              if(rq_write_lbp[index] == -1 and rq_read_lbp[index] != -1):
                  rq_write_lbp[index] = rq_read_lbp[index]
                  rq_write_lbp_previous[index] = rq_read_lbp[index]
              elif(rq_write_lbp_previous[index] == -1 and rq_read_lbp[index] != -1):
                  rq_write_lbp_previous[index] = rq_read_lbp[index]
              end

              if(rq_write_lrd[index] == -1 and rq_read_lrd[index] != -1):
                  rq_write_lrd[index] = rq_read_lrd[index]
                  rq_write_lrd_previous[index] = rq_read_lrd[index]
              elif(rq_write_lrd_previous[index] == -1 and rq_read_lrd[index] != -1):
                  rq_write_lrd_previous[index] = rq_read_lrd[index]
              end

              if(rq_write_lbl[index] == -1 and rq_read_lbl[index] != -1):
                  rq_write_lbl[index] = rq_read_lbl[index]
                  rq_write_lbl_previous[index] = rq_read_lbl[index]
              elif(rq_write_lbl_previous[index] == -1 and rq_read_lbl[index] != -1):
                  rq_write_lbl_previous[index] = rq_read_lbl[index]
              end

              if(rq_write_lgn[index] == -1 and rq_read_lgn[index] != -1):
                  rq_write_lgn[index] = rq_read_lgn[index]
                  rq_write_lgn_previous[index] = rq_read_lgn[index]
              elif(rq_write_lgn_previous[index] == -1 and rq_read_lgn[index] != -1):
                  rq_write_lgn_previous[index] = rq_read_lgn[index]
              end

              if(rq_write_msc[index] == -1 and rq_read_msc[index] != -1):
                  rq_write_msc[index] = rq_read_msc[index]
                  rq_write_msc_previous[index] = rq_read_msc[index]
              elif(rq_write_msc_previous[index] == -1 and rq_read_msc[index] != -1):
                  rq_write_msc_previous[index] = rq_read_msc[index]
              end

              if(rq_write_mod[index] == -1 and rq_read_mod[index] != -1):
                  rq_write_mod[index] = rq_read_mod[index]
                  rq_write_mod_previous[index] = rq_read_mod[index]
              elif(rq_write_mod_previous[index] == -1 and rq_read_mod[index] != -1):
                  rq_write_mod_previous[index] = rq_read_mod[index]
              end

          end
          index = index + 1
      end
  end

  def rq_comm_set_var(var, value=0, gripper_socket="1"):
      socket_set_var(var, value, gripper_socket)
      return socket_read_byte_list(3, gripper_socket)
  end

  def rq_comm_set_pos_spe_for(pos=0, speed=0, force=0, gripper_socket="1"):
      socket_send_string("SET POS", gripper_socket)
      socket_send_byte(32, gripper_socket)
      socket_send_string(pos, gripper_socket)
      socket_send_byte(32, gripper_socket)
      socket_send_string("SPE", gripper_socket)
      socket_send_byte(32, gripper_socket)
      socket_send_string(speed, gripper_socket)
      socket_send_byte(32, gripper_socket)
      socket_send_string("FOR", gripper_socket)
      socket_send_byte(32, gripper_socket)
      socket_send_string(force, gripper_socket)
      socket_send_byte(10, gripper_socket)
      return socket_read_byte_list(3, gripper_socket)
  end

  def rq_comm_read_variables():
      index = 0

      while(index <= 3):
          socket = rq_index_to_socket(index)

          if(gripper_connected[index]):

              if(rq_read_act_req[index]):
                  rq_read_act[index] = socket_get_var("ACT", socket)
                  rq_read_act_req[index] = False
              end

              if(rq_read_gto_req[index]):
                  rq_read_gto[index] = socket_get_var("GTO", socket)
                  rq_read_gto_req[index] = False
              end

              if(rq_read_pre_req[index]):
                  rq_read_pre[index] = socket_get_var("PRE", socket)
                  rq_read_pre_req[index] = False
              end

              if(rq_read_pos_req[index]):
                  rq_read_pos[index] = socket_get_var("POS", socket)
                  rq_read_pos_req[index] = False
              end

              if(rq_read_spe_req[index]):
                  rq_read_spe[index] = socket_get_var("SPE", socket)
                  rq_read_spe_req[index] = False
              end

              if(rq_read_for_req[index]):
                  rq_read_for[index] = socket_get_var("FOR", socket)
                  rq_read_for_req[index] = False
              end

              if(rq_read_obj_req[index]):
                  rq_read_obj[index] = socket_get_var("OBJ", socket)
                  rq_read_obj_req[index] = False
              end

              if(rq_read_sta_req[index]):
                  rq_read_sta[index] = socket_get_var("STA", socket)
                  rq_read_sta_req[index] = False
              end

              if(rq_read_mod_req[index]):
                  rq_read_mod[index] = socket_get_var("MOD", socket)
                  rq_read_mod_req[index] = False
              end

              if(rq_read_flt_req[index]):
                  rq_read_flt[index] = socket_get_var("FLT",socket)
                  rq_read_flt_req[index] = False
              end

              if(rq_read_lbp_req[index]):
                  rq_read_lbp[index] = socket_get_var("LBP", socket)
                  rq_read_lbp_req[index] = False
              end

              if(rq_read_lrd_req[index]):
                  rq_read_lrd[index] = socket_get_var("LRD", socket)
                  rq_read_lrd_req[index] = False
              end

              if(rq_read_lbl_req[index]):
                  rq_read_lbl[index] = socket_get_var("LBL",socket)
                  rq_read_lbl_req[index] = False
              end

              if(rq_read_lgn_req[index]):
                  rq_read_lgn[index] = socket_get_var("LGN", socket)
                  rq_read_lgn_req[index] = False
              end

              if(rq_read_msc_req[index]):
                  rq_read_msc[index] = socket_get_var("MSC", socket)
                  rq_read_msc_req[index] = False
              end

              if(rq_read_cou_req[index]):
                  rq_read_cou[index] = socket_get_var("COU", socket)
                  rq_read_cou_req[index] = False
              end

              if(rq_read_ncy_req[index]):
                  rq_read_ncy[index] = socket_get_var("NCY", socket)
                  rq_read_ncy_req[index] = False
              end

              if(rq_read_dst_req[index]):
                  rq_read_dst[index] = socket_get_var("DST", socket)
                  rq_read_dst_req[index] = False
              end

              if(rq_read_pco_req[index]):
                  rq_read_pco[index] = socket_get_var("PCO", socket)
                  rq_read_pco_req[index] = False
              end
          end
          index = index + 1
      end
  end

  def rq_comm_read_constants():

      if(gripper_connected[0]):
          while(rq_read_snu_1 == rq_string_initial_value):
              socket_send_string("GET SNU", "1")
              rq_read_snu_1 = socket_read_string("1")
          end

          while(rq_read_fwv_1 == rq_string_initial_value):
              socket_send_string("GET FWV", "1")
              rq_read_fwv_1 = socket_read_string("1")
          end

          while(rq_read_ver_1 == rq_string_initial_value):
              socket_send_string("GET VER", "1")
              rq_read_ver_1 = socket_read_string("1")
          end
      end

      if(gripper_connected[1]):
          while(rq_read_snu_2 == rq_string_initial_value):
              socket_send_string("GET SNU", "2")
              rq_read_snu_2 = socket_read_string("2")
          end

          while(rq_read_fwv_2 == rq_string_initial_value):
              socket_send_string("GET FWV", "2")
              rq_read_fwv_2 = socket_read_string("2")
          end

          while(rq_read_ver_2 == rq_string_initial_value):
              socket_send_string("GET VER", "2")
              rq_read_ver_2 = socket_read_string("2")
          end
      end

      if(gripper_connected[2]):
          while(rq_read_snu_3 == rq_string_initial_value):
              socket_send_string("GET SNU", "3")
              rq_read_snu_3 = socket_read_string("3")
          end

          while(rq_read_fwv_3 == rq_string_initial_value):
              socket_send_string("GET FWV", "3")
              rq_read_fwv_3 = socket_read_string("3")
          end

          while(rq_read_ver_3 == rq_string_initial_value):
              socket_send_string("GET VER", "3")
              rq_read_ver_3 = socket_read_string("3")
          end
      end

      if(gripper_connected[3]):
          while(rq_read_snu_4 == rq_string_initial_value):
              socket_send_string("GET SNU", "4")
              rq_read_snu_4 = socket_read_string("4")
          end

          while(rq_read_fwv_4 == rq_string_initial_value):
              socket_send_string("GET FWV", "4")
              rq_read_fwv_4 = socket_read_string("4")
          end

          while(rq_read_ver_4 == rq_string_initial_value):
              socket_send_string("GET VER", "4")
              rq_read_ver_4 = socket_read_string("4")
          end
      end
  end

  def rq_comm_write_variables():
      index = 0

      while(index <= 3):
          socket = rq_index_to_socket(index)

          if(gripper_connected[index]):

              if(rq_write_act_request[index]):
                  if(is_ack(rq_comm_set_var("ACT", rq_write_act[index], socket))):
                      rq_write_act_previous[index] = rq_write_act[index]
                      rq_write_act_request[index] = False
                  end
              end

              if(rq_write_gto_request[index]):
                  if(is_ack(rq_comm_set_var("GTO", rq_write_gto[index], socket))):
                      rq_write_gto_previous[index] = rq_write_gto[index]
                      rq_write_gto_request[index] = False
                  end
              end

              if(rq_write_atr_request[index]):
                  if(is_ack(rq_comm_set_var("ATR", rq_write_atr[index], socket))):
                      rq_write_atr_previous[index] = rq_write_atr[index]
                      rq_write_atr_request[index] = False
                  end
              end

              if(rq_write_ard_request[index]):
                  if(is_ack(rq_comm_set_var("ARD", rq_write_ard[index], socket))):
                      rq_write_ard_previous[index] = rq_write_ard[index]
                      rq_write_ard_request[index] = False
                  end
              end

              if(rq_write_pos_request[index]):
                  if(is_ack(rq_comm_set_pos_spe_for(rq_write_pos[index], rq_write_spe[index], rq_write_for[index], socket))):
                      rq_write_pos_previous[index] = rq_write_pos[index]
                      rq_write_spe_previous[index] = rq_write_spe[index]
                      rq_write_for_previous[index] = rq_write_for[index]
                      rq_write_pos_request[index] = False
                  end
              end

              if(rq_write_lbp_request[index]):
                  if(is_ack(rq_comm_set_var("LBP", rq_write_lbp[index], socket))):
                      rq_write_lbp_previous[index] = rq_write_lbp[index]
                      rq_write_lbp_request[index] = False
                  end
              end

              if(rq_write_lrd_request[index]):
                  if(is_ack(rq_comm_set_var("LRD", rq_write_lrd[index], socket))):
                      rq_write_lrd_previous[index] = rq_write_lrd[index]
                      rq_write_lrd_request[index] = False
                  end
              end

              if(rq_write_lbl_request[index]):
                  if(is_ack(rq_comm_set_var("LBL", rq_write_lbl[index], socket))):
                      rq_write_lbl_previous[index] = rq_write_lbl[index]
                      rq_write_lbl_request[index] = False
                  end
              end

              if(rq_write_lgn_request[index]):
                  if(is_ack(rq_comm_set_var("LGN", rq_write_lgn[index], socket))):
                      rq_write_lgn_previous[index] = rq_write_lgn[index]
                      rq_write_lgn_request[index] = False
                  end
              end

              if(rq_write_msc_request[index]):
                  if(is_ack(rq_comm_set_var("MSC", rq_write_msc[index], socket))):
                      rq_write_msc_previous[index] = rq_write_msc[index]
                      rq_write_msc_request[index] = False
                  end
              end

              if(rq_write_mod_request[index]):
                  if(is_ack(rq_comm_set_var("MOD", rq_write_mod[index], socket))):
                      rq_write_mod_previous[index] = rq_write_mod[index]
                      rq_write_mod_request[index] = False
                  end
              end
          end
          index = index + 1
      end
  end

  def rq_activate(gripper_socket="1"):
      if (not rq_is_gripper_activated(gripper_socket)):
          rq_reset(gripper_socket)

          while(not rq_get_var("ACT", 1, gripper_socket) == 0 or not rq_get_var("STA", 1, gripper_socket) == 0):
              rq_reset(gripper_socket)
              sleep(0.008)
          end

          rq_set_var("ACT",1, gripper_socket)
      end
  end

  def rq_activate_and_wait(gripper_socket="1"):
      if (not rq_is_gripper_activated(gripper_socket)):
          rq_activate(gripper_socket)
          sleep(1.0)

          while(not rq_get_var("ACT", 1, gripper_socket) == 1 or not rq_get_var("STA", 1, gripper_socket) == 3):
              sleep(0.1)
          end

          sleep(0.5)
      end
  end

  def rq_activate_all_grippers(reset=False):
      if(gripper_connected[0]):
          rq_reset_and_activate("1", reset)
      end

      if(gripper_connected[1]):
          rq_reset_and_activate("2", reset)
      end

      if(gripper_connected[2]):
          rq_reset_and_activate("3", reset)
      end

      if(gripper_connected[3]):
          rq_reset_and_activate("4", reset)
      end
  end

  def rq_reset_and_activate(gripper_socket="1", reset=False):
      if(reset):
          rq_reset(gripper_socket)
          rq_activate_and_wait(gripper_socket)
      elif(not rq_is_gripper_activated(gripper_socket)):
          rq_activate_and_wait(gripper_socket)
      end
  end

  def rq_reset(gripper_socket="1"):
      rq_set_var("ACT", 0, gripper_socket)
      rq_set_var("ATR", 0, gripper_socket)

      while(not rq_get_var("ACT", 1, gripper_socket) == 0 or not rq_get_var("STA", 1, gripper_socket) == 0):
          rq_set_var("ACT", 0, gripper_socket)
          rq_set_var("ATR", 0, gripper_socket)
          sleep(0.008)
      end

      sleep(0.5)
  end

  def rq_auto_release_open_and_wait(gripper_socket="1"):
      rq_set_var("ATR",0, gripper_socket)
      rq_set_var("ARD",0, gripper_socket)
      rq_set_var("ACT",1, gripper_socket)
      sleep(0.1)
      rq_set_var("ATR",1, gripper_socket)

      rq_wait_autorelease_completed(gripper_socket)
  end

  def rq_auto_release_close_and_wait(gripper_socket="1"):
      rq_set_var("ATR",0, gripper_socket)
      rq_set_var("ARD",1, gripper_socket)
      rq_set_var("ACT",1, gripper_socket)
      sleep(0.1)
      rq_set_var("ATR",1, gripper_socket)

      rq_wait_autorelease_completed(gripper_socket)
  end

  def rq_wait_autorelease_completed(gripper_socket="1"):
      remainingRetries = 20
      gFLT = rq_get_var("FLT", 2, gripper_socket)

      while(not is_FLT_autorelease_in_progress(gFLT) and remainingRetries > 0):
          remainingRetries = remainingRetries - 1
          gFLT = rq_get_var("FLT", 2, gripper_socket)
          sleep(0.1)
      end

      remainingRetries = 100
      gFLT = rq_get_var("FLT", 2, gripper_socket)

      while(not is_FLT_autorelease_completed(gFLT) and remainingRetries > 0):
          remainingRetries = remainingRetries - 1
          gFLT = rq_get_var("FLT", 2, gripper_socket)
          sleep(0.1)
      end
  end

  def rq_set_force(force, gripper_socket="1"):
      force = floor(scale(force, [0, 255], [0.0, 255.0]))
      rq_set_var("FOR", force, gripper_socket)
  end

  def rq_set_speed(speed, gripper_socket="1"):
      speed = floor(scale(speed, [0, 255], [0.0, 255.0]))
      rq_set_var("SPE", speed, gripper_socket)
  end

  def rq_open(gripper_socket="1"):
      rq_move(0, gripper_socket)
  end

  def rq_close(gripper_socket="1"):
      rq_move(255, gripper_socket)
  end

  def rq_open_and_wait(gripper_socket="1"):
      rq_move_and_wait(0, gripper_socket)
  end

  def rq_close_and_wait(gripper_socket="1"):
      rq_move_and_wait(255, gripper_socket)
  end

  def rq_move(pos, gripper_socket="1"):
      rq_set_pos(pos, gripper_socket)
      rq_go_to(gripper_socket)
  end

  def rq_move_and_wait(pos, gripper_socket="1"):
      rq_move(pos, gripper_socket)

      while (not rq_is_motion_complete(gripper_socket)):
          # wait for motion completed
          sleep(0.008)
      end
  end

  def rq_wait_for_pos_request(pos, gripper_socket="1"):
      gPRE = rq_get_var("PRE", 3, gripper_socket)

      while (gPRE != pos):
          rq_set_var("POS", pos, gripper_socket)
          sleep(0.008)
          gPRE = rq_get_var("PRE", 3, gripper_socket)
      end
  end

  def rq_wait_pos_spe_for_request(pos, speed, force, gripper_socket="1"):
      gPRE = rq_get_var("PRE", 3, gripper_socket)

      while (gPRE != pos):
          rq_set_pos_spe_for_var(pos, speed, force, gripper_socket)
          sleep(0.008)
          gPRE = rq_get_var("PRE", 3, gripper_socket)
      end
  end

  def rq_wait_for_pos(pos, gripper_socket="1"):
      rq_wait_for_pos_request(pos, gripper_socket)

      # Wait for the gripper motion to complete
      while (not rq_is_motion_complete(gripper_socket)):
          # wait for motion completed
          sleep(0.008)
          rq_set_var("GTO", 1, gripper_socket)
      end
  end

  def rq_wait(gripper_socket="1"):
      # Wait for the gripper motion to complete
      while (not rq_is_motion_complete(gripper_socket)):
          sleep(0.008)
          # The following patch is for Robotiq's Camera issue when communication is lost, but not the activation
          # the communication driver reset the GTO bit
          rq_set_var("GTO", 1, gripper_socket)
      end
  end

  def rq_wait_for_object_detected(gripper_socket="1"):
      # Wait the object detection
      while (not rq_is_object_detected(gripper_socket)):
          sleep(0.008)
      end
  end

  # set the position
  def rq_set_pos(pos, gripper_socket="1"):
      pos = floor(scale(pos, [0, 255], [0.0, 255.0]))
      rq_set_var("POS", pos, gripper_socket)
      rq_wait_for_pos_request(pos, gripper_socket)
  end

  def rq_set_pos_spd_for(pos, speed, force, gripper_socket="1"):
      pos = floor(scale(pos, [0, 255], [0.0, 255.0]))
      speed = floor(scale(speed, [0, 255], [0.0, 255.0]))
      force = floor(scale(force, [0, 255], [0.0, 255.0]))

      rq_set_pos_spe_for_var(pos, speed, force, gripper_socket)
  end

  def rq_set_gripper_max_current_mA(current_mA, gripper_socket="1"):
      current = floor(current_mA / 10)

      rq_set_var("MSC", current, gripper_socket)
      current_read = rq_get_var("MSC", 1, gripper_socket)

      while(current_read != current):
          rq_set_var("MSC", current, gripper_socket)
          current_read = rq_get_var("MSC", 1, gripper_socket)
      end
  end

  def rq_set_gripper_mode(mode, gripper_socket="1"):
      rq_set_var("MOD", mode, gripper_socket)
  end

  def rq_set_gripper_max_cur(current_mA, gripper_socket="1"):
      rq_set_gripper_max_current_mA(current_mA, gripper_socket)
  end

  def rq_get_gripper_max_current_mA(gripper_socket="1"):
      current = rq_get_var("MSC", 1, gripper_socket)

      if(current == -1):
          current_mA = current
      else:
          current_mA = current * 10
      end

      return current_mA
  end

  def rq_get_gripper_max_cur(gripper_socket="1"):
      return rq_get_gripper_max_current_mA(gripper_socket)
  end

  def rq_set_max_current_for_all_grippers():
      current_mA = rq_get_max_current_mA()

      if(gripper_connected[0]):
          rq_set_gripper_max_current_mA(current_mA, "1")
      end

      if(gripper_connected[1]):
          rq_set_gripper_max_current_mA(current_mA, "2")
      end

      if(gripper_connected[2]):
          rq_set_gripper_max_current_mA(current_mA, "3")
      end

      if(gripper_connected[3]):
          rq_set_gripper_max_current_mA(current_mA, "4")
      end
  end

  def rq_get_max_current_mA():
      max_current_mA = 0

      if(rq_current_limit_enabled):
          nb_connected_grippers = rq_get_nb_connected_grippers()

          if(nb_connected_grippers == 1):
              max_current_mA = 600
          elif(nb_connected_grippers > 1):
              max_current_mA = 450
          end
      else:

      end

      return max_current_mA
  end

  def rq_get_nb_connected_grippers():
      nb_connected_grippers = 0

      if(gripper_connected[0]):
          nb_connected_grippers = nb_connected_grippers + 1
      end

      if(gripper_connected[1]):
          nb_connected_grippers = nb_connected_grippers + 1
      end

      if(gripper_connected[2]):
          nb_connected_grippers = nb_connected_grippers + 1
      end

      if(gripper_connected[3]):
          nb_connected_grippers = nb_connected_grippers + 1
      end

      return nb_connected_grippers
  end

  def rq_list_of_bytes_to_value(list_of_bytes):
      value = -1

      # response list length
      if (list_of_bytes[0] == 1):
          value = list_of_bytes[1] - 48
      elif (list_of_bytes[0] == 2):
          value = (list_of_bytes[1] - 48) * 10 + (list_of_bytes[2] - 48)
      elif (list_of_bytes[0] == 3):
          value = (list_of_bytes[1] - 48) * 100 + (list_of_bytes[2] - 48) * 10 + (list_of_bytes[3] - 48)
      end

      return value
  end

  def rq_is_motion_complete(gripper_socket="1"):
      gOBJ = rq_get_var("OBJ", 1, gripper_socket)
      sleep(0.008)
      return is_OBJ_gripper_at_position(gOBJ) or is_OBJ_object_detected(gOBJ)
  end

  def rq_is_gripper_activated(gripper_socket="1"):
      gSTA = rq_get_var("STA", 1, gripper_socket)
      sleep(0.008)
      return is_STA_gripper_activated(gSTA)
  end

  def rq_is_object_detected(gripper_socket="1"):
      gOBJ = rq_get_var("OBJ", 1, gripper_socket)
      sleep(0.008)
      return is_OBJ_object_detected(gOBJ)
  end

  def rq_current_pos(gripper_socket="1"):
      gPOS = rq_get_var("POS", 1, gripper_socket)
      sleep(0.008)
      return gPOS
  end

  def rq_motor_current(gripper_socket="1"):
      rq_current = rq_get_var("COU", 1, gripper_socket)
      sleep(0.008)
      return rq_current * 10
  end

  def rq_print_connected_grippers():
      if(gripper_connected[0]):
          textmsg("Gripper 1 : ", "connected and socket open.")
      end

      if (gripper_connected[1]):
          textmsg("Gripper 2 : ", "connected and socket open.")
      end

      if (gripper_connected[2]):
          textmsg("Gripper 3 : ", "connected and socket open.")
      end

      if (gripper_connected[3]):
          textmsg("Gripper 4 : ", "connected and socket open.")
      end
  end

  def rq_print_gripper_fault_code(gripper_socket="1"):
      gFLT = rq_get_var("FLT", 2, gripper_socket)

      if(is_FLT_no_fault(gFLT)):
          textmsg("Gripper Fault : ", "No Fault (0x00)")
      elif (is_FLT_action_delayed(gFLT)):
          textmsg("Gripper Fault : ", "Priority Fault: Action delayed, initialization must be completed prior to performing the action (0x05)")
      elif (is_FLT_not_activated(gFLT)):
          textmsg("Gripper Fault : ", "Priority Fault: The activation bit must be set prior to performing the action (0x07)")
      elif (is_FLT_over_temperature(gFLT)):
          textmsg("Gripper Fault : ", "Minor Fault: Maximum operating temperature exceeded (≥ 85°C internally), let cool down (below 80°C) (0x08)")
      elif (is_FLT_no_communication(gFLT)):
          textmsg("Gripper Fault : ", "Minor Fault: No communication during at least 1 second (0x09)")
      elif (is_FLT_under_voltage(gFLT)):
          textmsg("Gripper Fault : ", "Major Fault: Under minimum operating voltage (0x0A)")
      elif (is_FLT_autorelease_in_progress(gFLT)):
          textmsg("Gripper Fault : ", "Major Fault: Automatic release in progress (0x0B)")
      elif (is_FLT_internal_fault(gFLT)):
          textmsg("Gripper Fault : ", "Major Fault: Internal fault; contact support@robotiq.com (0x0C)")
      elif (is_FLT_activation_error(gFLT)):
          textmsg("Gripper Fault : ", "Major Fault: Activation fault; verify that no interference or other error occurred (0x0D)")
      elif (is_FLT_overcurrent(gFLT)):
          textmsg("Gripper Fault : ", "Major Fault: Overcurrent triggered (0x0E)")
      elif (is_FLT_autorelease_completed(gFLT)):
          textmsg("Gripper Fault : ", "Major Fault: Automatic release completed (0x0F)")
      else:
          textmsg("Gripper Fault : ", "Unknown Fault")
      end
  end

  def rq_print_gripper_num_cycles(gripper_socket="1"):
      num_cycles = rq_get_var("NCY", 1, gripper_socket)

      if(num_cycles == -1):
          textmsg("Gripper Cycle Number : ", "Number of cycles is unreachable.")
      else:
          textmsg("Gripper Cycle Number : ", num_cycles)
      end
  end

  def rq_print_gripper_driver_state(gripper_socket="1"):
      driver_state = rq_get_var("DST", 1, gripper_socket)

      if(driver_state == 0):
          textmsg("Gripper Driver State : ", "RQ_STATE_INIT")
      elif(driver_state == 1):
          textmsg("Gripper Driver State : ", "RQ_STATE_LISTEN")
      elif(driver_state == 2):
          textmsg("Gripper Driver State : ", "RQ_STATE_READ_INFO")
      elif(driver_state == 3):
          textmsg("Gripper Driver State : ", "RQ_STATE_ACTIVATION")
      else:
          textmsg("Gripper Driver State : ", "RQ_STATE_RUN")
      end
  end

  def rq_print_gripper_serial_number(gripper_socket="1"):
      serial_number = rq_get_var_string("SNU", 1, gripper_socket)
      textmsg("Gripper Serial Number : ", serial_number)
  end

  def rq_print_gripper_firmware_version(gripper_socket="1"):
      firmware_version = rq_get_var_string("FWV", 1, gripper_socket)
      textmsg("Gripper Firmware Version : ", firmware_version)
  end

  def rq_print_gripper_driver_version(gripper_socket="1"):
      driver_version = rq_get_var_string("VER", 1, gripper_socket)
      textmsg("Gripper Driver Version : ", driver_version)
  end

  def rq_print_gripper_connection_state(gripper_socket="1"):
      connection_state = rq_get_var("PCO", 1, gripper_socket)

      if (connection_state == 0):
          textmsg("Gripper Connection State : ", "No connection problem detected")
      else:
          textmsg("Gripper Connection State : ", "Connection problem detected")
      end
  end

  # Returns True if list_of_bytes is [3, 'a', 'c', 'k']
  def is_ack(list_of_bytes):

      # list length is not 3
      if (list_of_bytes[0] != 3):
          return False
      end

      # first byte not is 'a'?
      if (list_of_bytes[1] != 97):
          return False
      end

      # first byte not is 'c'?
      if (list_of_bytes[2] != 99):
          return False
      end

      # first byte not is 'k'?
      if (list_of_bytes[3] != 107):
          return False
      end

      return True
  end

  # Returns True if list_of_bytes is not [3, 'a', 'c', 'k']
  def is_not_ack(list_of_bytes):
      if (is_ack(list_of_bytes)):
          return False
      else:
          return True
      end
  end

  def is_STA_gripper_activated (gSTA):
      if (gSTA == 3):
          return True
      end

      return False
  end

  def is_OBJ_object_detected (gOBJ):
      if (gOBJ == 1 or gOBJ == 2):
          return True
      end

      return False
  end

  def is_OBJ_gripper_at_position (gOBJ):
      if (gOBJ == 3):
          return True
      end

      return False
  end

  def is_not_OBJ_gripper_at_position (gOBJ):
      if (is_OBJ_gripper_at_position(gOBJ)):
          return False
      else:
          return True
      end
  end

  #### GTO Section ####
  def rq_stop(gripper_socket="1"):
      rq_set_var("GTO", 0, gripper_socket)
  end

  def rq_set_GTO_and_wait(value, gripper_socket="1"):
      rq_set_var("GTO" ,value, gripper_socket)
      while(not is_GTO(value, rq_get_var("GTO", 1, gripper_socket))):
        sleep(0.008)
      end
  end

  def rq_go_to(gripper_socket="1"):
      rq_set_var("GTO", 1, gripper_socket)
  end


  def is_GTO(goto_value, rGTO):
      return rGTO == goto_value
  end
  #### GTO Section ####

  def is_FLT_no_fault(gFLT):
      return gFLT == 0
  end

  def is_FLT_warning(gFLT):
      return gFLT >= 1 and gFLT <= 7
  end

  def is_FLT_faulted(gFLT):
      return gFLT >= 8
  end

  def is_FLT_action_delayed(gFLT):
      return gFLT == 5
  end

  def is_FLT_not_activated(gFLT):
      return gFLT == 7
  end

  def is_FLT_over_temperature(gFLT):
      return gFLT == 8
  end

  def is_FLT_no_communication(gFLT):
      return gFLT == 9
  end

  def is_FLT_under_voltage(gFLT):
      return gFLT == 10
  end

  def is_FLT_autorelease_in_progress(gFLT):
      return gFLT == 11
  end

  def is_FLT_internal_fault(gFLT):
      return gFLT == 12
  end

  def is_FLT_activation_error(gFLT):
      return gFLT == 13
  end

  def is_FLT_overcurrent(gFLT):
      return gFLT == 14
  end

  def is_FLT_autorelease_completed(gFLT):
      return gFLT == 15
  end

  def rq_set_var(var_name, var_value, gripper_socket="1"):
      index = rq_socket_to_index(gripper_socket)

      enter_critical

      if (var_name == "ACT"):
          rq_write_act[index] = var_value
          rq_write_act_request[index] = True
      elif (var_name == "GTO"):
          rq_write_gto[index] = var_value
          rq_write_gto_request[index] = True
      elif (var_name == "ATR"):
          rq_write_atr[index] = var_value
          rq_write_atr_request[index] = True
      elif (var_name == "ARD"):
          rq_write_ard[index] = var_value
          rq_write_ard_request[index] = True
      elif (var_name == "FOR"):
          rq_write_for[index] = var_value
          rq_write_pos_request[index] = True
      elif (var_name == "SPE"):
          rq_write_spe[index] = var_value
          rq_write_pos_request[index] = True
      elif (var_name == "POS"):
          rq_write_pos[index] = var_value
          rq_write_pos_request[index] = True
      elif (var_name == "LBP"):
          rq_write_lbp[index] = var_value
          rq_write_lbp_request[index] = True
      elif (var_name == "LRD"):
          rq_write_lrd[index] = var_value
          rq_write_lrd_request[index] = True
      elif (var_name == "LBL"):
          rq_write_lbl[index] = var_value
          rq_write_lbl_request[index] = True
      elif (var_name == "LGN"):
          rq_write_lgn[index] = var_value
          rq_write_lgn_request[index] = True
      elif (var_name == "MSC"):
          rq_write_msc[index] = var_value
          rq_write_msc_request[index] = True
      elif (var_name == "MOD"):
          rq_write_mod[index] = var_value
          rq_write_mod_request[index] = True
      end

      exit_critical

      if (var_name == "ACT"):
          while(rq_write_act_request[index]):
              sleep(0.008)
          end
      elif (var_name == "GTO"):
          while(rq_write_gto_request[index]):
              sleep(0.008)
          end
      elif (var_name == "ATR"):
          while(rq_write_atr_request[index]):
              sleep(0.008)
          end
      elif (var_name == "ARD"):
          while(rq_write_ard_request[index]):
              sleep(0.008)
          end
      elif (var_name == "FOR"):
          while(rq_write_pos_request[index]):
              sleep(0.008)
          end
      elif (var_name == "SPE"):
          while(rq_write_pos_request[index]):
              sleep(0.008)
          end
      elif (var_name == "POS"):
          while(rq_write_pos_request[index]):
              sleep(0.008)
          end
      elif (var_name == "LBP"):
          while(rq_write_lbp_request[index]):
              sleep(0.008)
          end
      elif (var_name == "LRD"):
          while(rq_write_lrd_request[index]):
              sleep(0.008)
          end
      elif (var_name == "LBL"):
          while(rq_write_lbl_request[index]):
              sleep(0.008)
          end
      elif (var_name == "LGN"):
          while(rq_write_lgn_request[index]):
              sleep(0.008)
          end
      elif (var_name == "MSC"):
          while(rq_write_msc_request[index]):
              sleep(0.008)
          end
      elif (var_name == "MOD"):
          while(rq_write_mod_request[index]):
              sleep(0.008)
          end
      end
  end

  def rq_set_pos_spe_for_var(pos, speed, force, gripper_socket="1"):
      index = rq_socket_to_index(gripper_socket)

      enter_critical

      rq_write_for[index] = force
      rq_write_spe[index] = speed
      rq_write_pos[index] = pos
      rq_write_pos_request[index] = True

      exit_critical
  end

  def rq_get_var(var_name, nbr_bytes, gripper_socket="1"):
      index = rq_socket_to_index(gripper_socket)
      var_value = -1

      if (var_name == "ACT"):
          enter_critical
          rq_read_act_req[index] = True
          exit_critical
          while(rq_read_act_req[index]):
              sleep(0.008)
          end
          var_value = rq_read_act[index]

      elif (var_name == "GTO"):
          enter_critical
          rq_read_gto_req[index] = True
          exit_critical
          while(rq_read_gto_req[index]):
              sleep(0.008)
          end
          var_value = rq_read_gto[index]

      elif (var_name == "FOR"):
          enter_critical
          rq_read_for_req[index] = True
          exit_critical
          while(rq_read_for_req[index]):
              sleep(0.008)
          end
          var_value = rq_read_for[index]

      elif (var_name == "SPE"):
          enter_critical
          rq_read_spe_req[index] = True
          exit_critical
          while(rq_read_spe_req[index]):
              sleep(0.008)
          end
          var_value = rq_read_spe[index]

      elif (var_name == "OBJ"):
          enter_critical
          rq_read_obj_req[index] = True
          exit_critical
          while(rq_read_obj_req[index]):
              sleep(0.008)
          end
          var_value = rq_read_obj[index]

      elif (var_name == "STA"):
          enter_critical
          rq_read_sta_req[index] = True
          exit_critical
          while(rq_read_sta_req[index]):
              sleep(0.008)
          end
          var_value = rq_read_sta[index]

      elif (var_name == "FLT"):
          enter_critical
          rq_read_flt_req[index] = True
          exit_critical
          while(rq_read_flt_req[index]):
              sleep(0.008)
          end
          var_value = rq_read_flt[index]

      elif (var_name == "POS"):
          enter_critical
          rq_read_pos_req[index] = True
          exit_critical
          while(rq_read_pos_req[index]):
              sleep(0.008)
          end
          var_value = rq_read_pos[index]

      elif (var_name == "PRE"):
          enter_critical
          rq_read_pre_req[index] = True
          exit_critical
          while(rq_read_pre_req[index]):
              sleep(0.008)
          end
          var_value = rq_read_pre[index]

      elif (var_name == "LBP"):
          enter_critical
          rq_read_lbp_req[index] = True
          exit_critical
          while(rq_read_lbp_req[index]):
              sleep(0.008)
          end
          var_value = rq_read_lbp[index]

      elif (var_name == "LRD"):
          enter_critical
          rq_read_lrd_req[index] = True
          exit_critical
          while(rq_read_lrd_req[index]):
              sleep(0.008)
          end
          var_value = rq_read_lrd[index]

      elif (var_name == "LBL"):
          enter_critical
          rq_read_lbl_req[index] = True
          exit_critical
          while(rq_read_lbl_req[index]):
              sleep(0.008)
          end
          var_value = rq_read_lbl[index]

      elif (var_name == "LGN"):
          enter_critical
          rq_read_lgn_req[index] = True
          exit_critical
          while(rq_read_lgn_req[index]):
              sleep(0.008)
          end
          var_value = rq_read_lgn[index]

      elif (var_name == "MSC"):
          enter_critical
          rq_read_msc_req[index] = True
          exit_critical
          while(rq_read_msc_req[index]):
              sleep(0.008)
          end
          var_value = rq_read_msc[index]

      elif (var_name == "MOD"):
          enter_critical
          rq_read_mod_req[index] = True
          exit_critical
          while(rq_read_mod_req[index]):
              sleep(0.008)
          end
          var_value = rq_read_mod[index]

      elif (var_name == "NCY"):
          enter_critical
          rq_read_ncy_req[index] = True
          exit_critical
          while(rq_read_ncy_req[index]):
              sleep(0.008)
          end
          var_value = rq_read_ncy[index]

      elif (var_name == "PCO"):
          enter_critical
          rq_read_pco_req[index] = True
          exit_critical
          while(rq_read_pco_req[index]):
              sleep(0.008)
          end
          var_value = rq_read_pco[index]

      elif (var_name == "DST"):
          enter_critical
          rq_read_dst_req[index] = True
          exit_critical
          while(rq_read_dst_req[index]):
              sleep(0.008)
          end
          var_value = rq_read_dst[index]

      end

      return var_value
  end

  def rq_get_var_string(var_name, nbr_bytes, gripper_socket="1"):
      index = rq_socket_to_index(gripper_socket)
      var_value = ""

      enter_critical

      if (var_name == "SNU"):
          if(gripper_socket == "1"):
              var_value = rq_read_snu_1
          elif(gripper_socket == "2"):
              var_value = rq_read_snu_2
          elif(gripper_socket == "3"):
              var_value = rq_read_snu_3
          elif(gripper_socket == "4"):
              var_value = rq_read_snu_4
          end
      elif (var_name == "FWV"):
          if(gripper_socket == "1"):
              var_value = rq_read_fwv_1
          elif(gripper_socket == "2"):
              var_value = rq_read_fwv_2
          elif(gripper_socket == "3"):
              var_value = rq_read_fwv_3
          elif(gripper_socket == "4"):
              var_value = rq_read_fwv_4
          end
      elif (var_name == "VER"):
          if(gripper_socket == "1"):
              var_value = rq_read_ver_1
          elif(gripper_socket == "2"):
              var_value = rq_read_ver_2
          elif(gripper_socket == "3"):
              var_value = rq_read_ver_3
          elif(gripper_socket == "4"):
              var_value = rq_read_ver_4
          end
      end

      exit_critical

      return var_value
  end

  def rq_is_object_validated(gripper_selected, gripper_socket="1"):
      if(gripper_selected):
          if(rq_is_object_detected(gripper_socket)):
              return True
          else:
              return False
          end
      else:
          return True
      end
  end

  ############################################
  # normalized functions (maps 0-100 to 0-255)
  ############################################
  def rq_set_force_norm(force_norm, gripper_socket="1"):
      force_gripper = norm_to_gripper(force_norm)
      rq_set_force(force_gripper, gripper_socket)
  end

  def rq_set_speed_norm(speed_norm, gripper_socket="1"):
      speed_gripper = norm_to_gripper(speed_norm)
      rq_set_speed(speed_gripper, gripper_socket)
  end

  def rq_move_norm(pos_norm, gripper_socket="1"):
      pos_gripper = norm_to_gripper(pos_norm)
      rq_move(pos_gripper, gripper_socket)
  end

  def rq_move_and_wait_norm(pos_norm, gripper_socket="1"):
      pos_gripper = norm_to_gripper(pos_norm)
      rq_move_and_wait(pos_gripper, gripper_socket)
  end

  def rq_set_pos_norm(pos_norm, gripper_socket="1"):
      pos_gripper = norm_to_gripper(pos_norm)
      rq_set_pos(pos_gripper, gripper_socket)
  end

  def rq_current_pos_norm(gripper_socket="1"):
      pos_gripper = rq_current_pos(gripper_socket)
      pos_norm = gripper_to_norm(pos_gripper)
      return pos_norm
  end

  def gripper_to_norm(value_gripper):
      value_norm = (value_gripper / 255) * 100
      return floor(value_norm)
  end

  def norm_to_gripper(value_norm):
      value_gripper = (value_norm / 100) * 255
      return ceil(value_gripper)
  end

  def rq_get_position():
      return rq_current_pos_norm()
  end

  def rq_gripper_led_on(gripper_socket="1"):
      rq_set_var("LBP",0, gripper_socket)
  end

  def rq_gripper_led_off(gripper_socket="1"):
      rq_set_var("LBP",1, gripper_socket)
      rq_set_var("LRD",0, gripper_socket)
      rq_set_var("LBL",0, gripper_socket)
      rq_set_var("LGN",0, gripper_socket)
  end

  def rq_gripper_led_force_red(gripper_socket="1"):
      rq_set_var("LBP",1, gripper_socket)
      rq_set_var("LRD",1, gripper_socket)
      rq_set_var("LBL",0, gripper_socket)
      rq_set_var("LGN",0, gripper_socket)
  end

  def rq_gripper_led_force_blue(gripper_socket="1"):
      rq_set_var("LBP",1, gripper_socket)
      rq_set_var("LRD",0, gripper_socket)
      rq_set_var("LBL",1, gripper_socket)
      rq_set_var("LGN",0, gripper_socket)
  end

  def rq_gripper_led_force_green(gripper_socket="1"):
      rq_set_var("LBP",1, gripper_socket)
      rq_set_var("LRD",0, gripper_socket)
      rq_set_var("LBL",0, gripper_socket)
      rq_set_var("LGN",1, gripper_socket)
  end

  def rq_gripper_led_force_purple(gripper_socket="1"):
      rq_set_var("LBP",1, gripper_socket)
      rq_set_var("LRD",1, gripper_socket)
      rq_set_var("LBL",1, gripper_socket)
      rq_set_var("LGN",0, gripper_socket)
  end

  ############################################
  # mm/inches functions
  ############################################
  gripper_closed_norm = [100, 100, 100, 100]
  gripper_open_norm = [0, 0, 0, 0]
  gripper_closed_mm = [0, 0, 0, 0]
  gripper_open_mm = [50, 50, 50, 50]

  def rq_current_pos_mm(gripper_socket=1):
      pos_gripper = rq_current_pos(gripper_socket)
      pos_mm = gripper_to_mm(pos_gripper, gripper_socket)
      return round_value_2_dec(pos_mm)
  end

  def rq_current_pos_inches(gripper_socket=1):
      pos_gripper = rq_current_pos(gripper_socket)
      pos_mm = gripper_to_mm(pos_gripper, gripper_socket)
      pos_in = pos_mm / 25.4
      return round_value_2_dec(pos_in)
  end

  def rq_move_mm(pos_mm, gripper_socket=1):
      pos_gripper = mm_to_gripper(pos_mm, gripper_socket)
      rq_move(pos_gripper, gripper_socket)
  end

  def rq_move_and_wait_mm(pos_mm, gripper_socket=1):
      pos_gripper = mm_to_gripper(pos_mm, gripper_socket)
      rq_move_and_wait(pos_gripper, gripper_socket)
  end

  def rq_move_inches(pos_in, gripper_socket=1):
      pos_mm = pos_in * 25.4
      rq_move_mm(pos_mm, gripper_socket)
  end

  def rq_move_and_wait_inches(pos_in, gripper_socket=1):
      pos_mm = pos_in * 25.4
      rq_move_and_wait_mm(pos_mm, gripper_socket)
  end

  def get_closed_norm(gripper_socket):
      return gripper_closed_norm[gripper_socket - 1]
  end

  def get_open_norm(gripper_socket):
      return gripper_open_norm[gripper_socket - 1]
  end

  def get_closed_mm(gripper_socket):
      return gripper_closed_mm[gripper_socket - 1]
  end

  def get_open_mm(gripper_socket):
      return gripper_open_mm[gripper_socket - 1]
  end

  def set_closed_norm(closed_norm, gripper_socket):
      gripper_closed_norm[gripper_socket - 1] = closed_norm
  end

  def set_open_norm(open_norm, gripper_socket):
      gripper_open_norm[gripper_socket - 1] = open_norm
  end

  def set_closed_mm(closed_mm, gripper_socket):
      gripper_closed_mm[gripper_socket - 1] = closed_mm
  end

  def set_open_mm(open_mm, gripper_socket):
      gripper_open_mm[gripper_socket - 1] = open_mm
  end

  def gripper_to_mm(value_gripper, gripper_socket):
      closed_norm = get_closed_norm(gripper_socket)
      open_norm = get_open_norm(gripper_socket)
      closed_mm = get_closed_mm(gripper_socket)
      open_mm = get_open_mm(gripper_socket)

      value_norm = (value_gripper / 255) * 100

      slope = (closed_mm - open_mm) / (closed_norm - open_norm)
      value_mm = slope * (value_norm - closed_norm) + closed_mm

      if (value_mm > open_mm):
          value_mm_limited = open_mm
      elif (value_mm < closed_mm):
          value_mm_limited = closed_mm
      else:
          value_mm_limited = value_mm
      end

      return value_mm_limited
  end

  def mm_to_gripper(value_mm, gripper_socket):
      closed_norm = get_closed_norm(gripper_socket)
      open_norm = get_open_norm(gripper_socket)
      closed_mm = get_closed_mm(gripper_socket)
      open_mm = get_open_mm(gripper_socket)

      slope = (closed_norm - open_norm) / (closed_mm - open_mm)
      value_norm = (value_mm - closed_mm) * slope + closed_norm

      value_gripper = value_norm * 255 / 100

      if (value_gripper > 255):
          value_gripper_limited = 255
      elif (value_gripper < 0):
          value_gripper_limited = 0
      else:
          value_gripper_limited = round_value(value_gripper)
      end

      return value_gripper_limited
  end

  def round_value(value):
      value_mod = value % 1

      if(value_mod < 0.5):
          return floor(value)
      else:
          return ceil(value)
      end
  end

  def round_value_2_dec(value):
      value_x_100 = value * 100
      value_x_100_rounded = round_value(value_x_100)
      return value_x_100_rounded / 100
  end

  def clear_socket_buffer(gripper_socket="1", read_timeout = 0.1):
      rq_comm_clear_socket_buffer_enabled[rq_socket_to_index(gripper_socket)] = True
  end

  def rq_gripper_id_to_ascii(gripper_id):
      if(gripper_id == "1"):
          return 57
      elif(gripper_id == "2"):
          return 50
      elif(gripper_id == "3"):
          return 51
      elif(gripper_id == "4"):
          return 52
      end
  end

  def scale(value, rawRange, scaledRange):
      def computeSlope(inputRange, outputRange):
          outputRangeDelta = outputRange[1] - outputRange[0]
          inputRangeDelta = inputRange[1] - inputRange[0]

          if (inputRangeDelta == 0):
              return 0
          else:
              return outputRangeDelta / inputRangeDelta
          end
      end

      def computeIntercept(slope, inputRange, outputRange):
          return outputRange[0] - (slope * inputRange[0])
      end

      def clipScaledValue(outputScaledValue, outputRange):
          if (outputRange[0] < outputRange[1]):
              return clipWhenLowerLimitIsLessThanHigher(outputScaledValue, outputRange)
          else:
              return clipWhenLowerLimitIsGreaterThanHigherLimit(outputScaledValue, outputRange)
          end
      end

      def clipWhenLowerLimitIsGreaterThanHigherLimit(outputScaledValue, outputRange):
          if (outputScaledValue < outputRange[1]):
              return outputRange[1]
          elif (outputScaledValue > outputRange[0]):
              return outputRange[0]
          else:
              return outputScaledValue
          end
      end

      def clipWhenLowerLimitIsLessThanHigher(outputScaledValue, outputRange):
          if (outputScaledValue < outputRange[0]):
              return outputRange[0]
          elif (outputScaledValue > outputRange[1]):
              return outputRange[1]
          else:
              return outputScaledValue
          end
      end

      slope = computeSlope(rawRange, scaledRange)
      intercept = computeIntercept(slope, rawRange, scaledRange)
      scaledValue = slope * value + intercept
      return clipScaledValue(scaledValue, scaledRange)
  end

  def limit(value, range):
      return scale(value, range, range)
  end


  rq_init_comm_if_connected(9, "1")
  rq_init_comm_if_connected(2, "2")
  rq_init_comm_if_connected(3, "3")
  rq_init_comm_if_connected(4, "4")
  rq_print_connected_grippers()
  rq_gripper_communication_thread = run rq_gripper_communication()
  set_closed_norm(100.0, 1)
  set_open_norm(0.0, 1)
  set_closed_mm(0.0, 1)
  set_open_mm(50.0, 1)
  set_closed_norm(100.0, 2)
  set_open_norm(0.0, 2)
  set_closed_mm(0.0, 2)
  set_open_mm(50.0, 2)
  set_closed_norm(100.0, 3)
  set_open_norm(0.0, 3)
  set_closed_mm(0.0, 3)
  set_open_mm(50.0, 3)
  set_closed_norm(100.0, 4)
  set_open_norm(0.0, 4)
  set_closed_mm(0.0, 4)
  set_open_mm(50.0, 4)
  rq_current_limit_enabled = False
  while(not rq_gripper_communication_thread_started):
      sleep(0.008)
  end
  # end: URCap Installation Node
  global start_p=p[.476445325383, .319648989491, .087962059422, .001631014108, -3.044455017533, .759623698847]
  global start_q=[3.6262218952178955, -1.0400421184352417, 1.7511833349811, -2.035672803918356, -1.9988163153277796, 2.1074979305267334]
  global clear_for_turn1_p=p[.488609844194, .434730459270, .178216608681, -2.886989623347, -.115415479293, .017142356595]
  global clear_for_turn1_q=[3.4924588203430176, -1.2129902702621003, 1.78257924715151, -2.207256933251852, -1.3281901518451136, -1.2923296133624476]
  global paketti_qr_p=p[-.021018894206, -.589950614873, .073343327060, -.099068556308, 3.003770378167, -.889003204106]
  global paketti_qr_q=[1.102047324180603, -1.0570516151240845, 2.442219320927755, -3.469151636163229, -1.29970628419985, -0.4644358793841761]
  global pickup_box_p=p[-.000490575086, -.525346496818, .154686878987, .074044090384, -3.139747310213, .001608022830]
  global pickup_box_q=[1.2317291498184204, -1.37679576993499, 2.0428269545184534, -2.2379008732237757, -1.572503391896383, -0.3866661230670374]
  global down_from_p=p[-.000476754745, -.525341762228, .154673509100, .074083662478, -3.139757887356, .001579523567]
  global down_to_p=p[-.000590824902, -.525483093308, -.006188474555, .074061717249, -3.139784973804, .001545937325]
  global Waypoint_1_from_p=p[-.000622529606, -.525517389986, -.006166014709, .074053462542, -3.139732157925, .001631720580]
  global Waypoint_1_to_p=p[-.000544296240, -.525404414544, .098834812701, .073944321263, -3.139749923830, .001624229300]
  $ 1 "BeforeStart"
  $ 2 "BeforeStartF"
  $ 3 "pcip≔'192.168.100.5'"
  global pcip="192.168.100.5"
  $ 4 "connection1≔False"
  global connection1=False
  $ 5 "Loop not connection1"
  while (not connection1):
    $ 6 "connection1≔socket_open(pcip,1201)"
    global connection1=socket_open(pcip,1201)
  end
  while (True):
    $ 7 "Robot Program"
    $ 8 "MoveJ"
    $ 9 "start" "breakAfter"
    movej(get_inverse_kin(start_p, qnear=start_q), a=1.3962634015954636, v=1.0471975511965976)
    $ 10 "loaded≔ False "
    global loaded=  False
    $ 11 "car_found≔ False "
    global car_found=  False
    $ 12 "socket_send_string('Enter car')"
    socket_send_string("Enter car")
    $ 13 "receive_srv≔socket_read_string(timeout=0)"
    global receive_srv=socket_read_string(timeout=0)
    $ 14 "socket_send_string('Enter packet')"
    socket_send_string("Enter packet")
    $ 15 "receive_srv1≔socket_read_string(timeout=0)"
    global receive_srv1=socket_read_string(timeout=0)
    $ 16 "socket_send_string(receive_srv)"
    socket_send_string(receive_srv)
    $ 17 "socket_send_string(receive_srv1)"
    socket_send_string(receive_srv1)
    $ 18 "'Cam locate to check for GoPiGo(s) in the loading zone'"
    # 'Cam locate to check for GoPiGo(s) in the loading zone'
    # begin: URCap Program Node
    #   Source: Robotiq_Wrist_Camera, 1.11.3.13312, Robotiq Inc.
    #   Type: Cam Locate
    $ 19 "Cam Locate"

    ###########################################
    #######VisionLocate node start########

    f=[0,0.0,0.0,0.0,0.0,0.0,0.0,0]
    object_location=p[0.0,0.0,0.0,0.0,0.0,0.0]
    feature_pose_to_restore_4791 = cal_new_rear
    movej([3.626171588897705, -1.0400675696185608, 1.7512033621417444, -2.0356890163817347, -1.9988740126239222, 2.1075141429901123])
    # Offset in translation only.
    snapshot_position_offset[3] = 0
    snapshot_position_offset[4] = 0
    snapshot_position_offset[5] = 0
    T_camera_in_flange = p[0, 0, 0, 0, 0, 0] # enlever une fois que l'enseignement du modele sera fait en faisant un movetool avec la pose de la camera dans le repere de la flange. Pour l'instant, on suppose que la camera est situee directement sur la flange.
    tool_4791 = get_T_in_base_from_flange(T_camera_in_flange)
    tool_4791 = pose_sub(tool_4791, snapshot_position_offset)
    snapshot_position = p[0.477009, 0.393883, 0.227503, 0.00149777, -3.04463, 0.75959]
    textmsg("expected snapshot position : ", snapshot_position)
    diff = pose_sub(tool_4791, snapshot_position)
    textmsg("diff = ", diff)
    is_at_snapshot_position = norm([diff[0], diff[1], diff[2]]) < 0.002
    is_at_snapshot_position = is_at_snapshot_position and (norm([diff[3], diff[4], diff[5]]) < 0.005)
    textmsg("is_at_snapshot_position = ", is_at_snapshot_position)
    is_snapshot_position_offset = norm(snapshot_position_offset) != 0
    is_at_snapshot_position = is_at_snapshot_position or ignore_snapshot_position
    if not(is_at_snapshot_position):
      popup("Robot is not at Snapshot Position. Add Move instruction to Snapshot Position before Camera Locate node.. Error code: [UCC-8]", warning = False, error = True)
      halt
    end
    f_4791 = xmlrpc_server.findmodel("contextName-4791", tool_4791[0], tool_4791[1], tool_4791[2], tool_4791[3], tool_4791[4], tool_4791[5])
    cam_locate_monitor.setFindModelResult("4791", f_4791)
    canSaveImage = True
    logging_service.publish("FIND_MODEL", f_4791)
    cam_locate_monitor.setCurrentObjectIndex("4791", 0)
    # begin: URCap Program Node
    #   Source: Robotiq_Wrist_Camera, 1.11.3.13312, Robotiq Inc.
    #   Type: Cam Locate Loop
    $ 20 "For object(s) found" "noBreak"
    object_teaching_location_4791 = p[0.5043233965545477, 0.4250833587958083, -0.023498287764681356, -0.012586435946725968, -3.133078542261244, -0.02614645774631396]
    feature_teaching_location_4791 = p[0.5043233965545477, 0.4250833587958083, -0.023498287764681356, -3.124637165397994, -0.02858001795767802, 0.012748500316914725]
    while (not cam_locate_monitor.isCaptureNeeded("4791")):
      poseAsArray = cam_locate_monitor.getCurrentObjectPoseAsArray("4791")
      current_object_location_4791 = p[poseAsArray[0], poseAsArray[1], poseAsArray[2], poseAsArray[3], poseAsArray[4], poseAsArray[5]]
      object_location = current_object_location_4791
      f[0] = cam_locate_monitor.getNumberOfObjectsFound("4791")
      f[1] = object_location[0]
      f[2] = object_location[1]
      f[3] = object_location[2]
      f[4] = object_location[3]
      f[5] = object_location[4]
      f[6] = object_location[5]
      f[7] = cam_locate_monitor.getCurrentObjectDetectionScore("4791")
      textmsg("current_object_location = ", current_object_location_4791)
      if (norm(snapshot_position_offset) != 0):
        current_object_location_4791 = pose_add(current_object_location_4791, snapshot_position_offset)
        textmsg("current_object_location after snapshot position offset = ", current_object_location_4791)
      end
      cal_new_rear = pose_trans(current_object_location_4791, pose_trans(pose_inv(object_teaching_location_4791), feature_teaching_location_4791))
      $ 21 "read_qr_pos≔pose_trans(cal_new_rear, p[0 ,0.12, -0.05, 0, 0.78, 3.14])" "noBreak"
      global read_qr_pos=pose_trans(cal_new_rear, p[0 ,0.12, -0.05, 0, 0.78, 3.14])
      $ 22 "MoveJ" "noBreak"
      $ 23 "read_qr_pos" "noBreak"
      movej(read_qr_pos, a=1.7453292519943295, v=1.7453292519943295)
      $ 24 "'Checking if the GoPiGo is present in the loading zone'" "noBreak"
      # 'Checking if the GoPiGo is present in the loading zone'
      # begin: URCap Program Node
      #   Source: Robotiq_Wrist_Camera, 1.11.3.13312, Robotiq Inc.
      #   Type: Scan Code
      $ 25 "Scan Code" "noBreak"

      ###########################################
      #######Scan code node start########

      canSaveImage = True
      socket_enabled_4651609 = False
      rq_find_code_4651609 = xmlrpc_server.findbarcode("contextName-37876", socket_enabled_4651609, "0.0.0.0", 0)
      nb_occurence_4651609 = rq_find_code_4651609[0]
      global rq_is_code_found = nb_occurence_4651609 > 0
      textmsg("rq_is_code_found = ", rq_is_code_found)
      i_4651609 = 0
      # begin: URCap Program Node
      #   Source: Robotiq_Wrist_Camera, 1.11.3.13312, Robotiq Inc.
      #   Type: If a code is found in Scan Code
      $ 26 "If a code is found" "noBreak"
      if (nb_occurence_4651609 > 0):
        while (i_4651609 < nb_occurence_4651609):
          rq_code_string_4651609 = xmlrpc_server.getbarcoderesult("contextName-37876", i_4651609)
          global rq_code_string = rq_code_string_4651609
          rq_code_quality = rq_find_code_4651609[2*i_4651609+1]
          rq_code_type = rq_find_code_4651609[2*i_4651609+2]
          textmsg("rq_code_string = ", rq_code_string)
          textmsg("rq_code_type = ", rq_code_type)
          i_4651609 = i_4651609 + 1
        end
        $ 27 "MoveJ" "noBreak"
        $ 28 "clear_for_turn1" "noBreak"
        movej(get_inverse_kin(pose_trans(cal_rear_table, pose_trans(p[.645600457556, -.015373178769, -.026410603389, 2.224347080471, -2.209846312426, -.027724163936], clear_for_turn1_p)), qnear=clear_for_turn1_q), a=1.7453292519943295, v=1.7453292519943295)
        $ 29 "If rq_code_string≟receive_srv" "noBreak"
        if (rq_code_string == receive_srv):
          $ 30 "'Cam locate for the packet(s)'" "noBreak"
          # 'Cam locate for the packet(s)'
          $ 31 "Loop  not loaded" "noBreak"
          while (  not  loaded):
            # begin: URCap Program Node
            #   Source: Robotiq_Wrist_Camera, 1.11.3.13312, Robotiq Inc.
            #   Type: Cam Locate
            $ 32 "Cam Locate" "noBreak"

            ###########################################
            #######VisionLocate node start########

            f=[0,0.0,0.0,0.0,0.0,0.0,0.0,0]
            object_location=p[0.0,0.0,0.0,0.0,0.0,0.0]
            feature_pose_to_restore_62702 = Calib_1
            if (cam_locate_monitor.isCaptureNeeded("62702")):
              movej([1.0477962493896484, -1.6324502430357875, 2.222819153462545, -2.6086260281004847, -1.3241484800921839, -0.46616870561708623])
              # Offset in translation only.
              snapshot_position_offset[3] = 0
              snapshot_position_offset[4] = 0
              snapshot_position_offset[5] = 0
              T_camera_in_flange = p[0, 0, 0, 0, 0, 0] # enlever une fois que l'enseignement du modele sera fait en faisant un movetool avec la pose de la camera dans le repere de la flange. Pour l'instant, on suppose que la camera est situee directement sur la flange.
              tool_62702 = get_T_in_base_from_flange(T_camera_in_flange)
              tool_62702 = pose_sub(tool_62702, snapshot_position_offset)
              snapshot_position = p[-0.0371989, -0.470642, 0.409203, 0.00138416, 3.03806, -0.788106]
              textmsg("expected snapshot position : ", snapshot_position)
              diff = pose_sub(tool_62702, snapshot_position)
              textmsg("diff = ", diff)
              is_at_snapshot_position = norm([diff[0], diff[1], diff[2]]) < 0.002
              is_at_snapshot_position = is_at_snapshot_position and (norm([diff[3], diff[4], diff[5]]) < 0.005)
              textmsg("is_at_snapshot_position = ", is_at_snapshot_position)
              is_snapshot_position_offset = norm(snapshot_position_offset) != 0
              is_at_snapshot_position = is_at_snapshot_position or ignore_snapshot_position
              if not(is_at_snapshot_position):
                popup("Robot is not at Snapshot Position. Add Move instruction to Snapshot Position before Camera Locate node.. Error code: [UCC-8]", warning = False, error = True)
                halt
              end
              f_62702 = xmlrpc_server.findmodel("contextName-62702", tool_62702[0], tool_62702[1], tool_62702[2], tool_62702[3], tool_62702[4], tool_62702[5])
              cam_locate_monitor.setFindModelResult("62702", f_62702)
              canSaveImage = True
              logging_service.publish("FIND_MODEL", f_62702)
              cam_locate_monitor.setCurrentObjectIndex("62702", 0)
            end
            # begin: URCap Program Node
            #   Source: Robotiq_Wrist_Camera, 1.11.3.13312, Robotiq Inc.
            #   Type: Cam Locate Loop
            $ 33 "For next object" "noBreak"
            object_teaching_location_62702 = p[-0.0053867573366070615, -0.47231310975799734, -0.006156285596003447, 0.005683687366064273, -3.140649904557625, 0.0016621203611247204]
            feature_teaching_location_62702 = p[-0.0053867573366070615, -0.47231310975799734, -0.006156285596003447, 2.179984864748392, 2.262050930447599, -0.002218470167007045]
            if (not cam_locate_monitor.isCaptureNeeded("62702")):
              poseAsArray = cam_locate_monitor.getCurrentObjectPoseAsArray("62702")
              current_object_location_62702 = p[poseAsArray[0], poseAsArray[1], poseAsArray[2], poseAsArray[3], poseAsArray[4], poseAsArray[5]]
              object_location = current_object_location_62702
              f[0] = cam_locate_monitor.getNumberOfObjectsFound("62702")
              f[1] = object_location[0]
              f[2] = object_location[1]
              f[3] = object_location[2]
              f[4] = object_location[3]
              f[5] = object_location[4]
              f[6] = object_location[5]
              f[7] = cam_locate_monitor.getCurrentObjectDetectionScore("62702")
              textmsg("current_object_location = ", current_object_location_62702)
              if (norm(snapshot_position_offset) != 0):
                current_object_location_62702 = pose_add(current_object_location_62702, snapshot_position_offset)
                textmsg("current_object_location after snapshot position offset = ", current_object_location_62702)
              end
              Calib_1 = pose_trans(current_object_location_62702, pose_trans(pose_inv(object_teaching_location_62702), feature_teaching_location_62702))
              $ 34 "MoveJ" "noBreak"
              $ 35 "paketti_qr" "noBreak"
              movej(get_inverse_kin(pose_trans(Calib_1, pose_trans(p[.471785258853, .022822739036, -.006662039349, -2.179984864755, -2.262050930455, .002218470161], paketti_qr_p)), qnear=paketti_qr_q), a=1.7453292519943295, v=1.7453292519943295)
              $ 36 "'Checking the Qr code in the packet(s)'" "noBreak"
              # 'Checking the Qr code in the packet(s)'
              # begin: URCap Program Node
              #   Source: Robotiq_Wrist_Camera, 1.11.3.13312, Robotiq Inc.
              #   Type: Scan Code
              $ 37 "Scan Code" "noBreak"

              ###########################################
              #######Scan code node start########

              canSaveImage = True
              socket_enabled_29393916 = False
              rq_find_code_29393916 = xmlrpc_server.findbarcode("contextName-2564", socket_enabled_29393916, "0.0.0.0", 0)
              nb_occurence_29393916 = rq_find_code_29393916[0]
              global rq_is_code_found = nb_occurence_29393916 > 0
              textmsg("rq_is_code_found = ", rq_is_code_found)
              i_29393916 = 0
              # begin: URCap Program Node
              #   Source: Robotiq_Wrist_Camera, 1.11.3.13312, Robotiq Inc.
              #   Type: If a code is found in Scan Code
              $ 38 "If a code is found" "noBreak"
              if (nb_occurence_29393916 > 0):
                while (i_29393916 < nb_occurence_29393916):
                  rq_code_string_29393916 = xmlrpc_server.getbarcoderesult("contextName-2564", i_29393916)
                  global rq_code_string = rq_code_string_29393916
                  rq_code_quality = rq_find_code_29393916[2*i_29393916+1]
                  rq_code_type = rq_find_code_29393916[2*i_29393916+2]
                  textmsg("rq_code_string = ", rq_code_string)
                  textmsg("rq_code_type = ", rq_code_type)
                  i_29393916 = i_29393916 + 1
                end
                $ 39 "If rq_code_string≟receive_srv1" "noBreak"
                if (rq_code_string == receive_srv1):
                  $ 40 "MoveJ" "noBreak"
                  $ 41 "pickup_box" "noBreak"
                  movej(get_inverse_kin(pose_trans(Calib_1, pose_trans(p[-.527758257806, -.030467615848, -.006662039354, -2.284063234482, 2.154944042682, -.000074196285], pickup_box_p)), qnear=pickup_box_q), a=1.7453292519943295, v=1.7453292519943295)
                  $ 42 "down" "noBreak"
                  movej(pose_add(get_target_tcp_pose(), pose_sub(down_to_p, down_from_p)), a=1.7453292519943295, v=1.7453292519943295)
                  # begin: URCap Program Node
                  #   Source: Robotiq_Grippers, 1.8.8.13523, Robotiq Inc.
                  #   Type: Vacuum
                  $ 43 "Vacuum Grip  (1)           " "noBreak"
                  if(not rq_is_gripper_connected("1")):
                      popup("A vacuum is not connected. ID: 1", "Vacuum Error", False, True, True)
                  end

                  rq_vacuum_grip_raw(True, 0, 60, 30, "1")

                      suction_completed = rq_wait_for_vacuum_object_suction_complete("1")
                      if(not suction_completed):
                          rq_set_var("GTO", 0, "1")
                      end

                  # end: URCap Program Node
                  $ 44 "Waypoint_1" "noBreak"
                  movej(pose_add(get_target_tcp_pose(), pose_sub(Waypoint_1_to_p, Waypoint_1_from_p)), a=1.7453292519943295, v=1.7453292519943295)
                  $ 45 "MoveJ" "noBreak"
                  $ 46 "start" "noBreak"
                  movej(get_inverse_kin(start_p, qnear=start_q), a=1.7453292519943295, v=1.7453292519943295)
                  $ 47 "drop_pos≔pose_trans(cal_new_rear, p[0, 0, -0.05, 0, 0, 3.14])" "noBreak"
                  global drop_pos= pose_trans (cal_new_rear, p[0, 0, -0.05, 0, 0, 3.14])
                  $ 48 "drop_pos" "noBreak"
                  movej(drop_pos, a=1.7453292519943295, v=1.7453292519943295)
                  # begin: URCap Program Node
                  #   Source: Robotiq_Grippers, 1.8.8.13523, Robotiq Inc.
                  #   Type: Vacuum
                  $ 49 "Vacuum Release  (1)           " "noBreak"
                  if(not rq_is_gripper_connected("1")):
                      popup("A vacuum is not connected. ID: 1", "Vacuum Error", False, True, True)
                  end

                  if(vacuumGripCheckThread1Running):
                      stopVacuumGripCheckThread(vacuumGripCheckThread1)
                      vacuumGripCheckThread1Running = False
                  end

                  rq_vacuum_release_raw(True, 100, 60, 255, 0.05, True, "1")

                  # end: URCap Program Node
                  $ 50 "Wait: 1.0" "noBreak"
                  sleep(1.0)
                  $ 51 "socket_send_string('Loaded')" "noBreak"
                  socket_send_string("Loaded")
                  $ 52 "loaded≔ True " "noBreak"
                  global loaded=  True
                  $ 53 "start" "noBreak"
                  movej(get_inverse_kin(start_p, qnear=start_q), a=1.7453292519943295, v=1.7453292519943295)
                end
              end
              # end: URCap Program Node
              # begin: URCap Program Node
              #   Source: Robotiq_Wrist_Camera, 1.11.3.13312, Robotiq Inc.
              #   Type: If no code found in Scan Code
              $ 54 "If no code found" "noBreak"
              if (nb_occurence_29393916 == 0):
                global rq_code_string = ""
                rq_code_quality = -1
                rq_code_type = -1
                $ 55 "'Optional'" "noBreak"
                # 'Optional'
                $ 56 "socket_send_string('paketti found, but not QR')" "noBreak"
                socket_send_string("paketti found, but not QR")
              end
              # end: URCap Program Node

              #######Scan Code node end########
              ###########################################

              # end: URCap Program Node
              cam_locate_monitor.incrementIndex("62702")
            end
            # end: URCap Program Node
            # begin: URCap Program Node
            #   Source: Robotiq_Wrist_Camera, 1.11.3.13312, Robotiq Inc.
            #   Type: If no object found in Camera Locate
            $ 57 "If no object found" "noBreak"
            if (not cam_locate_monitor.hasFoundObjects("62702")):
              f[0] = 0
              $ 58 "'Optional'" "noBreak"
              # 'Optional'
              $ 59 "socket_send_string('no paketti found')" "noBreak"
              socket_send_string("no paketti found")
            end
            # end: URCap Program Node
            # Restore feature pose
            Calib_1 = feature_pose_to_restore_62702

            #######VisionLocate node end########
            ###########################################

            # end: URCap Program Node
          end
        end
      end
      # end: URCap Program Node
      # begin: URCap Program Node
      #   Source: Robotiq_Wrist_Camera, 1.11.3.13312, Robotiq Inc.
      #   Type: If no code found in Scan Code
      $ 60 "If no code found" "noBreak"
      if (nb_occurence_4651609 == 0):
        global rq_code_string = ""
        rq_code_quality = -1
        rq_code_type = -1
        $ 61 "'Optional'" "noBreak"
        # 'Optional'
        $ 62 "socket_send_string('auto found, but not QR')" "noBreak"
        socket_send_string("auto found, but not QR")
      end
      # end: URCap Program Node

      #######Scan Code node end########
      ###########################################

      # end: URCap Program Node
      cam_locate_monitor.incrementIndex("4791")
    end
    # end: URCap Program Node
    # begin: URCap Program Node
    #   Source: Robotiq_Wrist_Camera, 1.11.3.13312, Robotiq Inc.
    #   Type: If no object found in Camera Locate
    $ 63 "If no object found" "noBreak"
    if (not cam_locate_monitor.hasFoundObjects("4791")):
      f[0] = 0
      $ 64 "'Optional'" "noBreak"
      # 'Optional'
      $ 65 "socket_send_string('auto not found')" "noBreak"
      socket_send_string("auto not found")
    end
    # end: URCap Program Node
    # Restore feature pose
    cal_new_rear = feature_pose_to_restore_4791

    #######VisionLocate node end########
    ###########################################

    # end: URCap Program Node
  end
end
